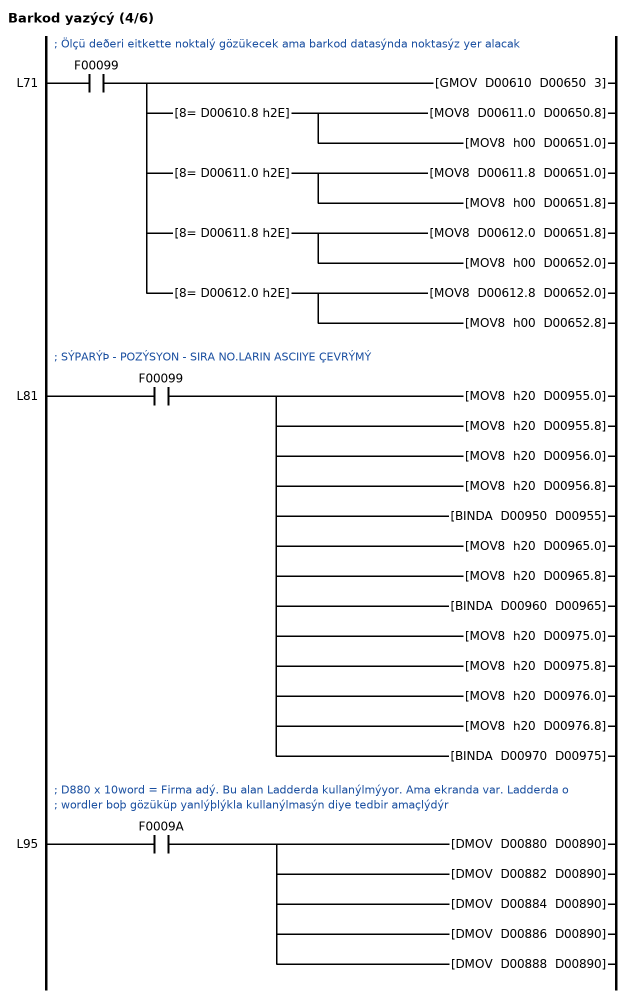
[picture p48: Barkod yazýcý rungs L71-L95]
// Ölçü deðeri eitkette noktalý gözükecek ama barkod datasýnda noktasýz yer alacak
; L71
LOAD      F00099
GMOV      D00610 D00650 3
MPUSH
AND8=     D00610.8 h2E
MOV8      D00611.0 D00650.8
MOV8      h00 D00651.0
MLOAD
AND8=     D00611.0 h2E
MOV8      D00611.8 D00651.0
MOV8      h00 D00651.8
MLOAD
AND8=     D00611.8 h2E
MOV8      D00612.0 D00651.8
MOV8      h00 D00652.0
MPOP
AND8=     D00612.0 h2E
MOV8      D00612.8 D00652.0
MOV8      h00 D00652.8
// SÝPARÝÞ - POZÝSYON - SIRA NO.LARIN ASCIIYE ÇEVRÝMÝ
; L81
LOAD      F00099
MOV8      h20 D00955.0
MOV8      h20 D00955.8
MOV8      h20 D00956.0
MOV8      h20 D00956.8
BINDA     D00950 D00955
MOV8      h20 D00965.0
MOV8      h20 D00965.8
BINDA     D00960 D00965
MOV8      h20 D00975.0
MOV8      h20 D00975.8
MOV8      h20 D00976.0
MOV8      h20 D00976.8
BINDA     D00970 D00975
// D880 x 10word = Firma adý. Bu alan Ladderda kullanýlmýyor. Ama ekranda var. Ladderda o wordler boþ gözüküp yanlýþlýkla kullanýlmasýn diye tedbir amaçlýdýr
; L95
LOAD      F0009A
DMOV      D00880 D00890
DMOV      D00882 D00890
DMOV      D00884 D00890
DMOV      D00886 D00890
DMOV      D00888 D00890

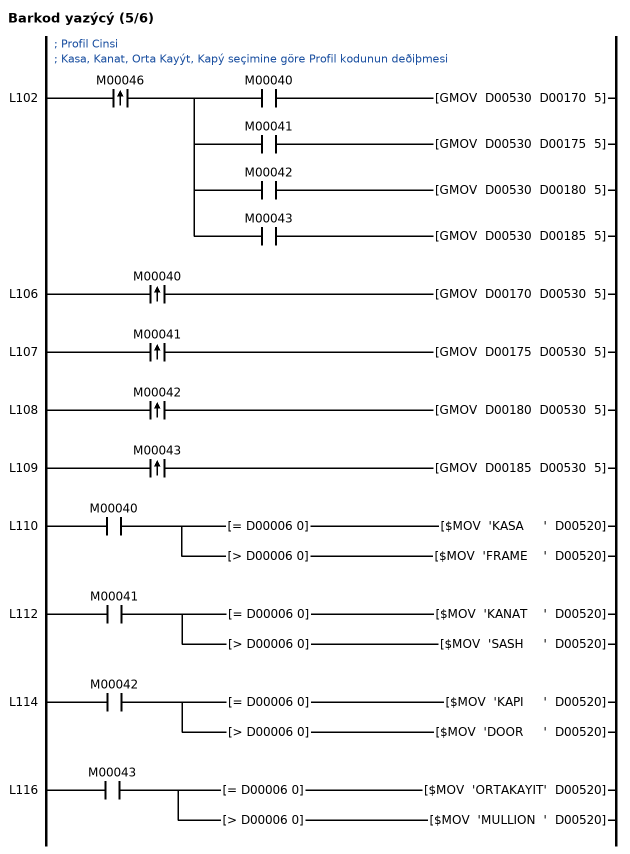
// Profil Cinsi
// Kasa, Kanat, Orta Kayýt, Kapý seçimine göre Profil kodunun deðiþmesi
; L102
LOADP     M00046
MPUSH
AND       M00040
GMOV      D00530 D00170 5
MLOAD
AND       M00041
GMOV      D00530 D00175 5
MLOAD
AND       M00042
GMOV      D00530 D00180 5
MPOP
AND       M00043
GMOV      D00530 D00185 5
; L106
LOADP     M00040
GMOV      D00170 D00530 5
; L107
LOADP     M00041
GMOV      D00175 D00530 5
; L108
LOADP     M00042
GMOV      D00180 D00530 5
; L109
LOADP     M00043
GMOV      D00185 D00530 5
; L110
LOAD      M00040
MPUSH
AND=      D00006 0
$MOV      'KASA     ' D00520
MPOP
AND>      D00006 0
$MOV      'FRAME    ' D00520
; L112
LOAD      M00041
MPUSH
AND=      D00006 0
$MOV      'KANAT    ' D00520
MPOP
AND>      D00006 0
$MOV      'SASH     ' D00520
; L114
LOAD      M00042
MPUSH
AND=      D00006 0
$MOV      'KAPI     ' D00520
MPOP
AND>      D00006 0
$MOV      'DOOR     ' D00520
; L116
LOAD      M00043
MPUSH
AND=      D00006 0
$MOV      'ORTAKAYIT' D00520
MPOP
AND>      D00006 0
$MOV      'MULLION  ' D00520

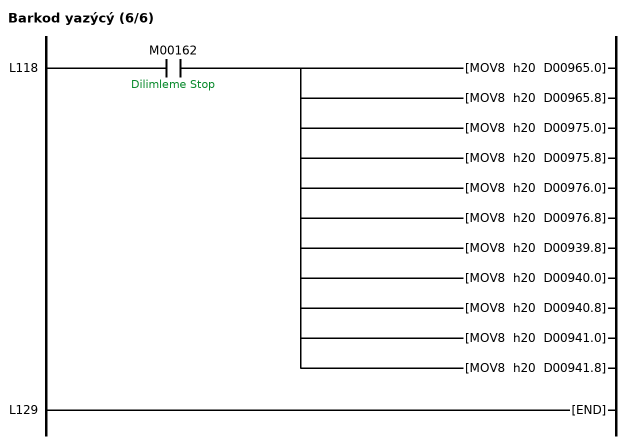
; L118
LOAD      M00162	// Dilimleme Stop
MOV8      h20 D00965.0
MOV8      h20 D00965.8
MOV8      h20 D00975.0
MOV8      h20 D00975.8
MOV8      h20 D00976.0
MOV8      h20 D00976.8
MOV8      h20 D00939.8
MOV8      h20 D00940.0
MOV8      h20 D00940.8
MOV8      h20 D00941.0
MOV8      h20 D00941.8
; L129
END

PROGRAM Teslimat Bilgileri (task: Scan Program)

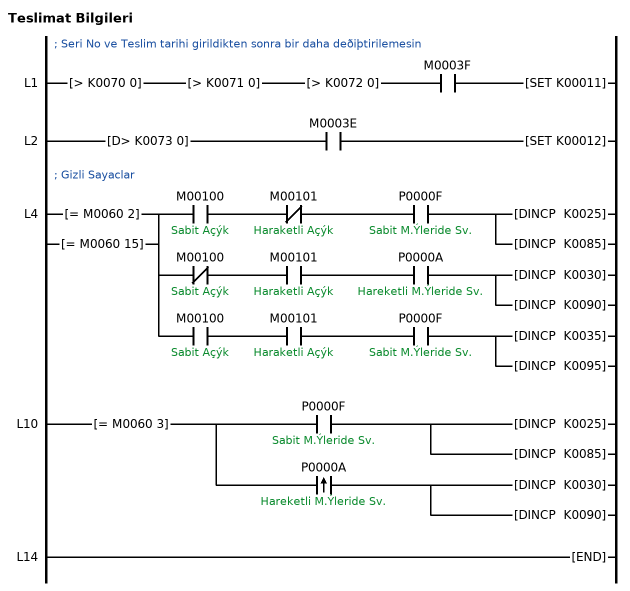
// Seri No ve Teslim tarihi girildikten sonra bir daha deðiþtirilemesin
; L1
LOAD>     K0070 0
AND>      K0071 0
AND>      K0072 0
AND       M0003F
SET       K00011
; L2
LOADD>    K0073 0
AND       M0003E
SET       K00012
// Gizli Sayaclar
; L4
LOAD=     M0060 2
OR=       M0060 15
MPUSH
AND       M00100	// Sabit Açýk
AND NOT   M00101	// Haraketli Açýk
AND       P0000F	// Sabit M.Ýleride Sv.
DINCP     K0025
DINCP     K0085
MLOAD
AND NOT   M00100	// Sabit Açýk
AND       M00101	// Haraketli Açýk
AND       P0000A	// Hareketli M.Ýleride Sv.
DINCP     K0030
DINCP     K0090
MPOP
AND       M00100	// Sabit Açýk
AND       M00101	// Haraketli Açýk
AND       P0000F	// Sabit M.Ýleride Sv.
DINCP     K0035
DINCP     K0095
; L10
LOAD=     M0060 3
MPUSH
AND       P0000F	// Sabit M.Ýleride Sv.
DINCP     K0025
DINCP     K0085
MPOP
ANDP      P0000A	// Hareketli M.Ýleride Sv.
DINCP     K0030
DINCP     K0090
; L14
END

VARIABLES AND COMMENTS (devices not used above)
M00900	BIT	tuning_start // tuning start
M00130	BIT	YErinde
M00163	BIT	Dilimleme Stop
M00133	BIT	Hareketli Kalibre
M00132	BIT	Sabit Kalibre
M00131	BIT	Boy Kalibre Baþla
M00420	BIT	Sabit Orijin
M00426	BIT	Sabit Preset
M00406	BIT	Sabit Preset Tamam
M00310	BIT	Sabit Reset
M00402	BIT	Sabit Meþgul
M00400	BIT	Sabit Orj.Tamam
M00410	BIT	Hareketli Orj.Tamam
M00436	BIT	Hareketli Preset
M00416	BIT	Hareketli Preset Tamam
M00320	BIT	Hareketli Reset
M00412	BIT	Hareketli Meþgul
M00430	BIT	Hareketli Orijin
M00437	BIT	Hareketli Jog
M00427	BIT	Sabit Jog
M00411	BIT	Hareketli Git Tamam
M00401	BIT	Sabit Git Tamam
M00404	BIT	sabit orjinde
M00414	BIT	hareketli orjinde
M00311	BIT	45 Kalibre-Sabit
M00314	BIT	90 Git-Sabit
M00316	BIT	Ayar+
M00317	BIT	Ayar-
M00312	BIT	90 Kalibre-Sabit
M00315	BIT	-90 Git (Kullanýlmýyor)-Sabit
M00313	BIT	45 Git-Sabit
M00318	BIT	Bitti
M00321	BIT	45 Kalibre-Hareketli
M00322	BIT	90 Kalibre-Hareketli
M00323	BIT	45 Git-Hareketli
M00324	BIT	90 Git-Hareketli
M00325	BIT	-90 Git (Kullanýlmýyor)-Hareketli
M00326	BIT	Ayar+
M00327	BIT	Ayar-
M00328	BIT	Bitti
M00438	BIT	Hareketli Jog
M00303	BIT	Metraj Kalibre Et
M00014	BIT	Hareketli Reset
M00319	BIT	Koruma
M00329	BIT	Koruma
M00210	BIT	Reçete-
M00211	BIT	Reçete+
M00212	BIT	Kayýt
M00213	BIT	Oku
M00154	BIT	Kasa
M00155	BIT	Kanat
M0011D	BIT	Uzun Boy
M00013	BIT	Kalibre Reset
M00158	BIT	Kasa Buton
M00159	BIT	Kanat Buton
M00450	BIT	Sabit Orijin Geri
M00451	BIT	Sabit Orijin Ýleri
M00452	BIT	Sabit Orijin Geri Yavaþ
M00460	BIT	Hareketli Orijin Geri
M00461	BIT	Harekelti Orijin Ýleri
M00462	BIT	Hareketli Orijin Geri Yavaþ
M00453	BIT	Sabit Preset
M00463	BIT	Hareketli Preset
M00407	BIT	Sabit Proks.
M00417	BIT	Hareketli Proks.
M00454	BIT	Sabit Ýleri
M00455	BIT	Sabit Geri
M00456	BIT	Sabit Jog
M00464	BIT	Hareketli Ýleri
M00465	BIT	Hareketli Geri
M00466	BIT	Hareketli Jog
M0001B	BIT	Sabit mt. Arýza
M0001C	BIT	Hareketli mt. Arýza
M00304	BIT	Katsayý -
M00128	BIT	Mengene Açý Kontrol
M00457	BIT	Ölçü Tamamlama
M00467	BIT	Ölçü Tamamlama
M00024	BIT	Boþluk toplama hareketi
D00072	WORD	Sabit Aþaðý yön durma noktasý düzeltme
D00076	WORD	Hareketli Aþaðý yön durma noktasý düzeltme
D00074	WORD	Hareketli Yukarý yön durma noktasý düzeltme
P00020	BIT	Pulse
P00022	BIT	Direction
M0003C	BIT	Seri No Kilidi